// TIA Portal V20 export
FUNCTION "IO映射" : Void   // FC4, LAD
{ S7_Optimized_Access := 'TRUE' }
// stored: SetENOAutomatically false
   VAR_TEMP
      LOOP : Int;
      Value : Byte;
      LOOP_1 : Int;
      Value_1 : Byte;
   END_VAR
BEGIN

REGION Network 1 (SCL)
   // 输入映射
   FOR #LOOP := 0 TO 10 BY 1 DO
       #Value := PEEK(area := 16#81, dbNumber := 0, byteOffset := #LOOP);
       POKE(area := 16#84,
            dbNumber := 12,
            byteOffset := #LOOP,
            value := #Value);
   END_FOR;
END_REGION

REGION Network 2 (SCL)
   // 输出映射
   FOR #LOOP_1 := 0 TO 8 BY 1 DO
       #Value_1 := PEEK(area := 16#84, dbNumber := 13, byteOffset := #LOOP_1);
       POKE(area := 16#82,
            dbNumber := 0,
            byteOffset := #LOOP_1,
            value := #Value_1);
   END_FOR;
END_REGION

REGION Network 3
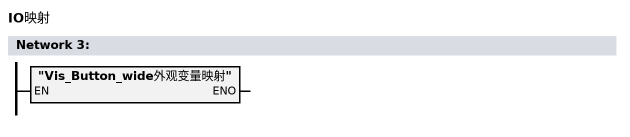
   RUNG wire#powerrail
      "Vis_Button_wide外观变量映射"()
   END_RUNG
   // the same network as SCL:
   "Vis_Button_wide外观变量映射"();
END_REGION
END_FUNCTION
